FUNCTION_BLOCK FB_VisionController EXTENDS FB_VisionCameraBase
VAR_INPUT
END_VAR
VAR_OUTPUT
END_VAR
VAR
END_VAR

METHOD ProcessImage
END_METHOD

END_FUNCTION_BLOCK

(* stored: Version 1.1.0.1
   POU FB_VisionController: Id {38653925-2c14-40fc-aead-2847ea230b56}, SpecialFunc None
   Method ProcessImage: Id {f3614d49-889b-4492-88a4-066783cb385b} *)
